// TIA Portal V20 export
TYPE "IB_P01_02_03_in_64bytes_struct"
// stored: Access Published, Namespace Global
   STRUCT
      Reserved : Byte;
      Sens_A : Bool;
      Sens_B : Bool;
      Sens_A_alrm : Bool;
      Sens_B_alrm : Bool;
      Motor_state_A : Bool;
      Motor_state_B : Bool;
      Reserved_1 : Bool;
      Reserved_2 : Bool;
      Fuse_err_A : Bool;
      Back_EMF_err_A : Bool;
      Thermal_err_mot_A : Bool;
      Thermal_err_ctrl_A : Bool;
      Lock_err_A : Bool;
      Unconnected_err_A : Bool;
      Reserved_3 : Bool;
      Reserved_4 : Bool;
      Fuse_err_B : Bool;
      Back_EMF_err_B : Bool;
      Thermal_err_mot_B : Bool;
      Thermal_err_ctrl_B : Bool;
      Lock_err_B : Bool;
      Unconnected_err_B : Bool;
      Reserved_5 : Bool;
      Reserved_6 : Bool;
      Digital_in_1 : Bool;   // NA for IB-P03
      Digital_in_2 : Bool;   // NA for IB-P03
      Digital_in_3 : Bool;   // NA for IB-P03
      Digital_in_4 : Bool;   // NA for IB-P03
      Reserved_7 : Bool;
      Reserved_8 : Bool;
      Reserved_9 : Bool;
      Reserved_10 : Bool;
      Register_Low_D0 : Byte;
      Register_High_D0 : Byte;
      Register_Low_D1 : Byte;
      Register_High_D1 : Byte;
      Register_Low_D2 : Byte;
      Register_High_D2 : Byte;
      Register_Low_D3 : Byte;
      Register_High_D3 : Byte;
      Register_Low_D4 : Byte;
      Register_High_D4 : Byte;
      Register_Low_D5 : Byte;
      Register_High_D5 : Byte;
      Register_Low_D6 : Byte;
      Register_High_D6 : Byte;
      Register_Low_D7 : Byte;
      Register_High_D7 : Byte;
      Register_Low_D8 : Byte;
      Register_High_D8 : Byte;
      Register_Low_D9 : Byte;
      Register_High_D9 : Byte;
      Register_Low_D10 : Byte;
      Register_High_D10 : Byte;
      Register_Low_D11 : Byte;
      Register_High_D11 : Byte;
      Register_Low_D12 : Byte;
      Register_High_D12 : Byte;
      Register_Low_D13 : Byte;
      Register_High_D13 : Byte;
      Register_Low_D14 : Byte;
      Register_High_D14 : Byte;
      Register_Low_D15 : Byte;
      Register_High_D15 : Byte;
      Life_time_mot_A_LL : Byte;
      Life_time_mot_A_LH : Byte;
      Life_time_mot_A_HL : Byte;
      Life_time_mot_A_HH : Byte;
      Life_time_mot_B_LL : Byte;
      Life_time_mot_B_LH : Byte;
      Life_time_mot_B_HL : Byte;
      Life_time_mot_B_HH : Byte;
      Current_mot_A : Byte;
      Current_mot_B : Byte;
      Voltage_mot_A : Byte;
      Voltage_mot_B : Byte;
      Reserved_11 : Array[0..13] of Byte;
   END_STRUCT;
END_TYPE
